(* IEC 61131-3 sources: wago_2pump_ebm_fans/PFC200_G2_2ETH_RS_CAN_DPS_T.device.xml.v3^/Plc Logic.plclogic.xml.v3^/Application.application.xml.v3^/TCPServer/DataFunc, 8 files *)

(* ---- getBathCalibrate.fn.st ---- *)
FUNCTION getBathCalibrate : STRING(300)
VAR_INPUT
	Bath:		POINTER TO Bath;
END_VAR
VAR
END_VAR

getBathCalibrate := '';
//
getBathCalibrate := CONCAT(getBathCalibrate, UINT_TO_STRING(Bath^.BathConfig.CalibrateInPressureSensorMIN));
getBathCalibrate := CONCAT(getBathCalibrate ,':');
//
getBathCalibrate := CONCAT(getBathCalibrate, UINT_TO_STRING(Bath^.BathConfig.CalibrateInPressureSensorDelta));
getBathCalibrate := CONCAT(getBathCalibrate ,':');
//
getBathCalibrate := CONCAT(getBathCalibrate, UINT_TO_STRING(Bath^.BathConfig.CalibrateOutPressureSensorMIN));
getBathCalibrate := CONCAT(getBathCalibrate ,':');
//
getBathCalibrate := CONCAT(getBathCalibrate, UINT_TO_STRING(Bath^.BathConfig.CalibrateOutPressureSensorDelta));

(* ---- getBathConf.fn.st ---- *)
FUNCTION getBathConf : STRING(300)
VAR_INPUT
	Bath:		POINTER TO Bath;
END_VAR
VAR
END_VAR

getBathConf := '';
//AdminMainRelay
getBathConf := CONCAT(getBathConf, UINT_TO_STRING(Bath^.BathConfig.AdminMainRelay));
getBathConf := CONCAT(getBathConf ,':');
//AdminPumpRelay
getBathConf := CONCAT(getBathConf, UINT_TO_STRING(Bath^.BathConfig.AdminPumpRelay));
getBathConf := CONCAT(getBathConf ,':');
//AdminFanRelay
getBathConf := CONCAT(getBathConf, UINT_TO_STRING(Bath^.BathConfig.AdminFanRelay));
getBathConf := CONCAT(getBathConf ,':');
//LiquidStepInterval
getBathConf := CONCAT(getBathConf, TIME_TO_STRING(Bath^.BathConfig.LiquidStepInterval));
getBathConf := CONCAT(getBathConf ,':');
//LiquidTargetTemp
getBathConf := CONCAT(getBathConf, UINT_TO_STRING(Bath^.BathConfig.LiquidTargetTemp));
getBathConf := CONCAT(getBathConf ,':');
//LiquidAlertTemp
getBathConf := CONCAT(getBathConf, UINT_TO_STRING(Bath^.BathConfig.LiquidAlertTemp));
getBathConf := CONCAT(getBathConf ,':');
//PressureStabilizeInterval
getBathConf := CONCAT(getBathConf, TIME_TO_STRING(Bath^.BathConfig.PressureStabilizeInterval));
getBathConf := CONCAT(getBathConf ,':');
//PressureStabilizeTarget
getBathConf := CONCAT(getBathConf, REAL_TO_STRING(Bath^.BathConfig.PressureStabilizeTarget));
getBathConf := CONCAT(getBathConf ,':');
//FanMinFreq
getBathConf := CONCAT(getBathConf, UINT_TO_STRING(Bath^.BathConfig.FanMinFreq));

(* ---- getBathStats.fn.st ---- *)
FUNCTION getBathStats : STRING(300)
VAR_INPUT
	Bath:		POINTER TO Bath;
END_VAR
VAR
END_VAR

getBathStats := '';
//Liquid in temp
getBathStats := CONCAT(getBathStats, INT_TO_STRING(REAL_TO_INT(Bath^.LiquidInTemp*100)));
getBathStats := CONCAT(getBathStats ,':');
//Liquid Out Temp
getBathStats := CONCAT(getBathStats, INT_TO_STRING(REAL_TO_INT(Bath^.LiquidOutTemp*100)));
getBathStats := CONCAT(getBathStats ,':');
//Pressure Incoming
getBathStats := CONCAT(getBathStats, UINT_TO_STRING(REAL_TO_UINT(Bath^.PressureIncoming*100)));
getBathStats := CONCAT(getBathStats ,':');
//Pressure Outgoing
getBathStats := CONCAT(getBathStats, UINT_TO_STRING(REAL_TO_UINT(Bath^.PressureOutgoing*100)));
getBathStats := CONCAT(getBathStats ,':');
//Freq
getBathStats := CONCAT(getBathStats, UINT_TO_STRING(REAL_TO_UINT(Bath^.Freq)));
getBathStats := CONCAT(getBathStats ,':');
//MainStatus
getBathStats := CONCAT(getBathStats, INT_TO_STRING(Bath^.MainStatus));
getBathStats := CONCAT(getBathStats ,':');
//TempStatus
getBathStats := CONCAT(getBathStats, INT_TO_STRING(Bath^.TempStatus));
getBathStats := CONCAT(getBathStats ,':');
//LevelStatus
getBathStats := CONCAT(getBathStats, INT_TO_STRING(Bath^.LevelStatus));
getBathStats := CONCAT(getBathStats ,':');
//MainRelayTripStatus
getBathStats := CONCAT(getBathStats, BOOL_TO_STRING(Bath^.MainRelayTripStatus));
getBathStats := CONCAT(getBathStats ,':');
//MainKMTripStatus
getBathStats := CONCAT(getBathStats, BOOL_TO_STRING(Bath^.MainKMTripStatus));
getBathStats := CONCAT(getBathStats ,':');
//PumpKMTripStatus
getBathStats := CONCAT(getBathStats, BOOL_TO_STRING(Bath^.PumpKMTripStatus));
getBathStats := CONCAT(getBathStats ,':');
//PumpCBTripStatus
getBathStats := CONCAT(getBathStats, BOOL_TO_STRING(Bath^.PumpCBTripStatus));
getBathStats := CONCAT(getBathStats ,':');
//ACCBTripStatus
getBathStats := CONCAT(getBathStats, BOOL_TO_STRING(Bath^.ACCBTripStatus));
getBathStats := CONCAT(getBathStats ,':');
//MainRelayStatus
getBathStats := CONCAT(getBathStats, BOOL_TO_STRING(Bath^.MainRelayStatus));
getBathStats := CONCAT(getBathStats ,':');
//MainKMStatus
getBathStats := CONCAT(getBathStats, BOOL_TO_STRING(Bath^.MainKMStatus));
getBathStats := CONCAT(getBathStats ,':');
//PumpKMStatus
getBathStats := CONCAT(getBathStats, BOOL_TO_STRING(Bath^.PumpKMStatus));

(* ---- getCalibrate.fn.st ---- *)
FUNCTION getCalibrate : STRING(500)
VAR_INPUT
END_VAR
VAR
	Bath1Conf : STRING(300);
	Bath2Conf : STRING(300);
END_VAR

getCalibrate := 'START:';
Bath1Conf := getBathCalibrate(Bath := ADR(GVL.Baths[0]));
getCalibrate := CONCAT(getCalibrate, Bath1Conf);
getCalibrate := CONCAT(getCalibrate, ':');
Bath2Conf := getBathCalibrate(Bath := ADR(GVL.Baths[1]));
getCalibrate := CONCAT(getCalibrate, Bath2Conf);

(* ---- getConf.fn.st ---- *)
FUNCTION getConf : STRING(500)
VAR_INPUT
END_VAR
VAR
	Bath1Conf : STRING(300);
	Bath2Conf : STRING(300);
END_VAR

getConf := 'START:';
Bath1Conf := getBathConf(Bath := ADR(GVL.Baths[0]));
getConf := CONCAT(getConf, Bath1Conf);
getConf := CONCAT(getConf, ':');
Bath2Conf := getBathConf(Bath := ADR(GVL.Baths[1]));
getConf := CONCAT(getConf, Bath2Conf);
getConf := CONCAT(getConf ,':');
//HighAirTemp
getConf := CONCAT(getConf, UINT_TO_STRING(PV.HighAirTemp));
getConf := CONCAT(getConf, ':END');

(* ---- getStats.fn.st ---- *)
FUNCTION getStats : STRING(500)
VAR_INPUT
END_VAR
VAR
	Bath1Stat : STRING(300);
	Bath2Stat : STRING(300);
END_VAR

getStats := 'START:';
Bath1Stat := getBathStats(Bath := ADR(GVL.Baths[0]));
getStats := CONCAT(getStats, Bath1Stat);
getStats := CONCAT(getStats, ':');
Bath2Stat := getBathStats(Bath := ADR(GVL.Baths[1]));
getStats := CONCAT(getStats, Bath2Stat);
getStats := CONCAT(getStats, ':');
getStats := CONCAT(getStats, UINT_TO_STRING(REAL_TO_UINT(GVL.ContainerAirTemp*100)));
getStats := CONCAT(getStats, ':');
getStats := CONCAT(getStats, UINT_TO_STRING(REAL_TO_UINT(GVL.ContainerAirHumi*100)));
getStats := CONCAT(getStats, ':');
getStats := CONCAT(getStats, UINT_TO_STRING(REAL_TO_UINT(GVL.CabinetAirTemp*100)));
getStats := CONCAT(getStats, ':');
getStats := CONCAT(getStats, UINT_TO_STRING(REAL_TO_UINT(GVL.CabinetAirHumi*100)));
getStats := CONCAT(getStats, ':END');

(* ---- updateCalibrate.fn.st ---- *)
FUNCTION updateCalibrate : STRING(150);
VAR_INPUT
	sString			: STRING(300);
END_VAR
VAR
	sSeparatorChar: STRING := ':';
	configArray		: ARRAY [0..8] OF STRING;
	i,j,configPosition: INT;

	configCheck : INT := 1;
END_VAR

j := 0;
configPosition := 0;

FOR i:= 0 TO LEN(sString) DO
	IF sString[i] = sSeparatorChar[0] THEN
		configArray[configPosition] := MID(sString, i-j+1, j);
		configPosition := configPosition + 1;
		j := i + 2;
	END_IF
END_FOR

configArray[configPosition] := MID(sString, i-j, j);

IF configPosition = 8 THEN
	PV.BathConfigs[0].CalibrateInPressureSensorMIN := STRING_TO_UINT(configArray[configCheck]);
	configCheck := configCheck +1;

	PV.BathConfigs[0].CalibrateInPressureSensorDelta := STRING_TO_UINT(configArray[configCheck]);
	configCheck := configCheck +1;

	PV.BathConfigs[0].CalibrateOutPressureSensorMIN := STRING_TO_UINT(configArray[configCheck]);
	configCheck := configCheck +1;

	PV.BathConfigs[0].CalibrateOutPressureSensorDelta := STRING_TO_UINT(configArray[configCheck]);
	configCheck := configCheck +1;

	PV.BathConfigs[1].CalibrateInPressureSensorMIN := STRING_TO_UINT(configArray[configCheck]);
	configCheck := configCheck +1;

	PV.BathConfigs[1].CalibrateInPressureSensorDelta := STRING_TO_UINT(configArray[configCheck]);
	configCheck := configCheck +1;

	PV.BathConfigs[1].CalibrateOutPressureSensorMIN := STRING_TO_UINT(configArray[configCheck]);
	configCheck := configCheck +1;

	PV.BathConfigs[1].CalibrateOutPressureSensorDelta := STRING_TO_UINT(configArray[configCheck]);
	configCheck := configCheck +1;

	GVL.Baths[0].BathConfig := PV.BathConfigs[0];
	GVL.Baths[1].BathConfig := PV.BathConfigs[1];

	updateCalibrate := 'SUCCESS';
ELSE
	updateCalibrate := 'FAIL';
END_IF

(* ---- updateConf.fn.st ---- *)
FUNCTION updateConf : STRING(150);
VAR_INPUT
	sString			: STRING(300);
END_VAR
VAR
	sSeparatorChar: STRING := ':';
	configArray		: ARRAY [0..19] OF STRING;
	i,j,configPosition: INT;

	configCheck : INT := 1;
END_VAR

j := 0;
configPosition := 0;

FOR i:= 0 TO LEN(sString) DO
	IF sString[i] = sSeparatorChar[0] THEN
		configArray[configPosition] := MID(sString, i-j+1, j);
		configPosition := configPosition + 1;
		j := i + 2;
	END_IF
END_FOR

configArray[configPosition] := MID(sString, i-j, j);

IF configPosition = 19 THEN
	IF STRING_TO_INT(configArray[configCheck]) = 0 THEN
		PV.BathConfigs[0].AdminMainRelay := ENUM_AdminRelayStatus.relayForceEnable;
	ELSIF STRING_TO_INT(configArray[configCheck]) = 1 THEN
		PV.BathConfigs[0].AdminMainRelay := ENUM_AdminRelayStatus.relayAutoEnable;
	ELSIF STRING_TO_INT(configArray[configCheck]) = 2 THEN
		PV.BathConfigs[0].AdminMainRelay := ENUM_AdminRelayStatus.relayForceDisable;
	END_IF

	configCheck := configCheck +1;

	IF STRING_TO_INT(configArray[configCheck]) = 0 THEN
		PV.BathConfigs[0].AdminPumpRelay := ENUM_AdminRelayStatus.relayForceEnable;
	ELSIF STRING_TO_INT(configArray[configCheck]) = 1 THEN
		PV.BathConfigs[0].AdminPumpRelay := ENUM_AdminRelayStatus.relayAutoEnable;
	ELSIF STRING_TO_INT(configArray[configCheck]) = 2 THEN
		PV.BathConfigs[0].AdminPumpRelay := ENUM_AdminRelayStatus.relayForceDisable;
	END_IF

	configCheck := configCheck +1;

	IF STRING_TO_INT(configArray[configCheck]) = 0 THEN
		PV.BathConfigs[0].AdminFanRelay := ENUM_AdminRelayStatus.relayForceEnable;
	ELSIF STRING_TO_INT(configArray[configCheck]) = 1 THEN
		PV.BathConfigs[0].AdminFanRelay := ENUM_AdminRelayStatus.relayAutoEnable;
	ELSIF STRING_TO_INT(configArray[configCheck]) = 2 THEN
		PV.BathConfigs[0].AdminFanRelay := ENUM_AdminRelayStatus.relayForceDisable;
	END_IF

	configCheck := configCheck +1;

	PV.BathConfigs[0].LiquidStepInterval := STRING_TO_TIME(configArray[configCheck]);
	configCheck := configCheck +1;

	PV.BathConfigs[0].LiquidTargetTemp := STRING_TO_UINT(configArray[configCheck]);
	configCheck := configCheck +1;

	PV.BathConfigs[0].LiquidAlertTemp := STRING_TO_UINT(configArray[configCheck]);
	configCheck := configCheck +1;

	PV.BathConfigs[0].PressureStabilizeInterval := STRING_TO_TIME(configArray[configCheck]);
	configCheck := configCheck +1;

	PV.BathConfigs[0].PressureStabilizeTarget := STRING_TO_REAL(configArray[configCheck]);
	configCheck := configCheck +1;

	PV.BathConfigs[0].FanMinFreq := STRING_TO_UINT(configArray[configCheck]);
	configCheck := configCheck +1;

	IF STRING_TO_INT(configArray[configCheck]) = 0 THEN
		PV.BathConfigs[1].AdminMainRelay := ENUM_AdminRelayStatus.relayForceEnable;
	ELSIF STRING_TO_INT(configArray[configCheck]) = 1 THEN
		PV.BathConfigs[1].AdminMainRelay := ENUM_AdminRelayStatus.relayAutoEnable;
	ELSIF STRING_TO_INT(configArray[configCheck]) = 2 THEN
		PV.BathConfigs[1].AdminMainRelay := ENUM_AdminRelayStatus.relayForceDisable;
	END_IF
	configCheck := configCheck +1;

	IF STRING_TO_INT(configArray[configCheck]) = 0 THEN
		PV.BathConfigs[1].AdminPumpRelay := ENUM_AdminRelayStatus.relayForceEnable;
	ELSIF STRING_TO_INT(configArray[configCheck]) = 1 THEN
		PV.BathConfigs[1].AdminPumpRelay := ENUM_AdminRelayStatus.relayAutoEnable;
	ELSIF STRING_TO_INT(configArray[configCheck]) = 2 THEN
		PV.BathConfigs[1].AdminPumpRelay := ENUM_AdminRelayStatus.relayForceDisable;
	END_IF
	configCheck := configCheck +1;

	IF STRING_TO_INT(configArray[configCheck]) = 0 THEN
		PV.BathConfigs[1].AdminFanRelay := ENUM_AdminRelayStatus.relayForceEnable;
	ELSIF STRING_TO_INT(configArray[configCheck]) = 1 THEN
		PV.BathConfigs[1].AdminFanRelay := ENUM_AdminRelayStatus.relayAutoEnable;
	ELSIF STRING_TO_INT(configArray[configCheck]) = 2 THEN
		PV.BathConfigs[1].AdminFanRelay := ENUM_AdminRelayStatus.relayForceDisable;
	END_IF
	configCheck := configCheck +1;

	PV.BathConfigs[1].LiquidStepInterval := STRING_TO_TIME(configArray[configCheck]);
	configCheck := configCheck +1;

	PV.BathConfigs[1].LiquidTargetTemp := STRING_TO_UINT(configArray[configCheck]);
	GVL.Baths[0].LiquidIncreaseMax := STRING_TO_REAL(configArray[configCheck]);
	GVL.Baths[1].LiquidIncreaseMax := STRING_TO_REAL(configArray[configCheck]);
	GVL.Baths[0].LiquidDecreaseMax := STRING_TO_REAL(configArray[configCheck]);
	GVL.Baths[1].LiquidDecreaseMax := STRING_TO_REAL(configArray[configCheck]);
	configCheck := configCheck +1;

	PV.BathConfigs[1].LiquidAlertTemp := STRING_TO_UINT(configArray[configCheck]);
	configCheck := configCheck +1;

	PV.BathConfigs[1].PressureStabilizeInterval := STRING_TO_TIME(configArray[configCheck]);
	configCheck := configCheck +1;

	PV.BathConfigs[1].PressureStabilizeTarget := STRING_TO_REAL(configArray[configCheck]);
	configCheck := configCheck +1;

	PV.BathConfigs[1].FanMinFreq := STRING_TO_UINT(configArray[configCheck]);
	configCheck := configCheck +1;

	PV.HighAirTemp := STRING_TO_UINT(configArray[configCheck]);

	GVL.Baths[0].BathConfig := PV.BathConfigs[0];
	GVL.Baths[1].BathConfig := PV.BathConfigs[1];

	updateConf := 'SUCCESS';
ELSE
	updateConf := 'FAIL';
END_IF
